{attribute 'GeneratedUsingTerminal: AT2050-0501-0024'}
{attribute addProperty BoxType "AT2050-0501-0024"}
{attribute addProperty Id "A_0084_AT2050_5500_0017_AT2050_5500AT2050_01D6DEDF80"}
{attribute addProperty CRC "2541302476"}
{attribute addProperty Size "80"}
TYPE A_0072_AT2050_0501_0024_AT2050_0501_977932CC EXTENDS AT2050_86175B41 :
STRUCT
	{attribute addProperty Name "A_0084_AT2050_5500_0017_AT2050_5500"}
	A_0084_AT2050_5500_0017_AT2050_5500 : AT2050_01D6DEDF;
END_STRUCT
END_TYPE

(* stored: Version 1.2.0.0, ProductVersion 3.1.4024.9
   DUT A_0072_AT2050_0501_0024_AT2050_0501_977932CC: Id {9bdb4cf5-a85e-4634-bd40-9a95359621ca} *)
